Staubli VAL3: DisplayPt.pgx

public program DisplayPt(trsf x_trLoc, num x_nRaw)
  local trsf l_trLoc
begin
  // This program display the coordinates of a location on the userPage
  //
  // Input Param
  //  x_pLoc  : Location to display
  //  x_nRaw  : Raw on which the coordinates must be displayed
  //
  // Output param
  //
  call type(4,x_nRaw,"X Y Z :")
  call type(12,x_nRaw,toString(".2",x_trLoc.x))
  call type(21,x_nRaw,toString(".2",x_trLoc.y))
  call type(30,x_nRaw,toString(".2",x_trLoc.z))
  call type(4,x_nRaw+1,"RxRyRz:")
  call type(12,x_nRaw+1,toString(".2",x_trLoc.rx))
  call type(21,x_nRaw+1,toString(".2",x_trLoc.ry))
  call type(30,x_nRaw+1,toString(".2",x_trLoc.rz))
end
